FUNCTION_BLOCK PUBLIC PAEEMotorFreq2D EXTENDS PAEEMotorFreqCtrl
VAR_INPUT
END_VAR
VAR_OUTPUT
END_VAR
VAR
	_PAPointMatInOut1 : PAPoint(THIS^);
	_PAPointMatInOut2 : PAPoint(THIS^);
	_DirectionLeft : BOOL;
	_ReqDirectionLeft : BOOL;
	_ToggleAllowed : BOOL;
END_VAR

{attribute 'monitoring' := 'call'}
//{attribute 'TcRpcEnable'}
PROPERTY PUBLIC DirectionLeft : BOOL
GET // PUBLIC
DirectionLeft := _DirectionLeft;
END_GET
SET // PUBLIC
_DirectionLeft := DirectionLeft;
Root.OnPropertyChangedBool(THIS^, 50, _DirectionLeft);
END_SET
END_PROPERTY

METHOD FB_init : BOOL
VAR_INPUT
	bInitRetains : BOOL; // if TRUE, the retain variables are initialized (warm start / cold start)
	bInCopyCode : BOOL;  // if TRUE, the instance afterwards gets moved into the copy code (online change)
	parent : IACComponent;
END_VAR
AddPoint(_PAPointMatInOut1);
AddPoint(_PAPointMatInOut2);
END_METHOD

METHOD FB_postinit
VAR_INPUT
		root : IACVariobatch;	
END_VAR
SUPER^.FB_postinit(root);  
root.OnPropertyChangedBool(THIS^, 50, _DirectionLeft);
root.OnPropertyChangedBool(THIS^, 51, _ReqDirectionLeft);
END_METHOD

METHOD PUBLIC HasPointReachedOffPosition : BOOL
VAR_INPUT
	point : IACPoint;
END_VAR
IF point = PAPointMatInOut1 OR point = PAPointMatInOut2 THEN
	HasPointReachedOffPosition := NOT _RunState;
ELSE
	HasPointReachedOffPosition := FALSE;
END_IF
END_METHOD

METHOD PUBLIC HasPointReachedOnPosition : BOOL
VAR_INPUT
	point : IACPoint;
END_VAR
IF point = PAPointMatInOut1 THEN
	HasPointReachedOnPosition :=    ((NOT _DirectionLeft) 
										AND _RunState 
										AND (   (_Speed >= (_ReqSpeed - 0.001))
											 OR (_Speed >= (_DesiredSpeed - 0.001)))
									 )
								OR _DirectionLeft; // Fungiert als Eingangspunkt
ELSIF point = PAPointMatInOut2 THEN
	HasPointReachedOnPosition := 	(_DirectionLeft 
										AND _RunState 
										AND (   (_Speed >= (_ReqSpeed - 0.001))
											 OR (_Speed >= (_DesiredSpeed - 0.001)))
									 )
								OR NOT _DirectionLeft; // Fungiert als Eingangspunkt
ELSE
	HasPointReachedOnPosition := FALSE;
END_IF
END_METHOD

METHOD PUBLIC InvokeSetterBool
VAR_INPUT
	PropertyID : INT;
	PropertyValue : BOOL;
END_VAR
SUPER^.InvokeSetterBool(PropertyID, PropertyValue);
IF PropertyID = 50 THEN
	DirectionLeft := PropertyValue;
ELSIF PropertyID = 51 THEN	
	ReqDirectionLeft := PropertyValue;
END_IF
END_METHOD

METHOD PUBLIC IsEnabledTurnOnLeft : BOOL
VAR_INPUT
END_VAR
END_METHOD

METHOD PUBLIC IsEnabledTurnOnRight : BOOL
VAR_INPUT
END_VAR
END_METHOD

METHOD OnInitMemory
VAR_INPUT
	root : IACVariobatch;
END_VAR
RegisterProperty(root, 50, GCL.cSizeBYTE); //DirectionLeft
RegisterProperty(root, 51, GCL.cSizeBYTE); //ReqDirectionLeft
SUPER^.OnInitMemory(root);
END_METHOD

PROPERTY PUBLIC PAPointMatInOut1 : IACPoint
GET // PUBLIC
PAPointMatInOut1 := _PAPointMatInOut1;
END_GET
END_PROPERTY

PROPERTY PUBLIC PAPointMatInOut2 : IACPoint
GET // PUBLIC
PAPointMatInOut2 := _PAPointMatInOut2;
END_GET
END_PROPERTY

{attribute 'monitoring' := 'call'}
//{attribute 'TcRpcEnable'}
PROPERTY PUBLIC ReqDirectionLeft : BOOL
GET // PUBLIC
ReqDirectionLeft := _ReqDirectionLeft;
END_GET
SET // PUBLIC
_ReqDirectionLeft := ReqDirectionLeft;
Root.OnPropertyChangedBool(THIS^, 51, _ReqDirectionLeft);
IF Root.InSimulation THEN
	DirectionLeft := _ReqDirectionLeft;
END_IF
END_SET
END_PROPERTY

{attribute 'monitoring' := 'call'}
//{attribute 'TcRpcEnable'}
PROPERTY PUBLIC ToggleAllowed : BOOL
GET // PUBLIC
ToggleAllowed := _ToggleAllowed;
END_GET
SET // PUBLIC
_ToggleAllowed := ToggleAllowed;
END_SET
END_PROPERTY

METHOD PUBLIC TurnOnLeft
VAR_INPUT
END_VAR
END_METHOD

METHOD PUBLIC TurnOnRight
VAR_INPUT
END_VAR
END_METHOD

METHOD PUBLIC TurnOnWithSpeed
VAR_INPUT
END_VAR
END_METHOD

END_FUNCTION_BLOCK

(* stored: Version 1.1.0.1, ProductVersion 3.1.4024.6
   POU PAEEMotorFreq2D: Id {48f8e403-c1e5-4f25-915b-859ff11263ce}, SpecialFunc None
   Property DirectionLeft: Id {61ae9675-b877-4012-9877-4f55053bb8cd}
   Get Get: Id {ab51ae8e-092f-495e-971b-d436360d7d86}
   Set Set: Id {22da2eed-9936-4c72-bc7a-e6371c4fdd15}
   Method FB_init: Id {1a0d4860-71cb-4c98-ae1e-860ae42e16cf}
   Method FB_postinit: Id {08db1755-b296-41cb-88fc-411631b56700}
   Method HasPointReachedOffPosition: Id {6eff92e2-0f72-49d0-9cb0-7ebf94c01c7c}
   Method HasPointReachedOnPosition: Id {7eb4fe3d-ce5c-4ed4-bdfe-6ccd3d48c5c6}
   Method InvokeSetterBool: Id {0864a1a0-76f3-4cf5-a812-3bcf475ad3d8}
   Method IsEnabledTurnOnLeft: Id {40e12c0e-e94b-4e49-a4c9-93cf967ac42e}
   Method IsEnabledTurnOnRight: Id {5d87ff20-227a-451c-861e-5d6410eaafe2}
   Method OnInitMemory: Id {0cf9a302-4224-4ebd-b78c-f579f0f6b148}
   Property PAPointMatInOut1: Id {f2d1768f-e37e-4f83-8bd6-ad234d2c2a45}
   Get Get: Id {26acfe4a-ed9d-49d2-9670-13749866b44e}
   Property PAPointMatInOut2: Id {5ee328e9-f028-4855-931a-04635492f3bb}
   Get Get: Id {fffc46f0-9ebe-4350-81ae-8ad47efa6209}
   Property ReqDirectionLeft: Id {9c42cad5-2d9f-4305-85ce-f5e3ef8812bb}
   Get Get: Id {15288849-38ed-4a42-b6bd-f932da215aab}
   Set Set: Id {eed12a0e-af90-47f1-ad72-caadcf3714dd}
   Property ToggleAllowed: Id {a02fdccd-5882-43fb-8719-dee60d3cab93}
   Get Get: Id {a4acced5-1596-405e-8eda-f3541750a6e3}
   Set Set: Id {818694be-aa7b-43fa-86e6-06b2dd427cde}
   Method TurnOnLeft: Id {167cdc7b-4826-414e-a7fe-fc1f82ab4586}
   Method TurnOnRight: Id {a7cc28ca-57f1-4285-a508-cecb3f3d84e7}
   Method TurnOnWithSpeed: Id {b170feb8-2c8e-46fe-98d9-64c00406da8d} *)
